INTERFACE ITcoCustomizedDialogFormat

METHOD WithCaption : ITcoCustomizedDialogAnswer
VAR_INPUT
	inCaption : STRING(255);
END_VAR
END_METHOD

METHOD WithImage : ITcoCustomizedDialogAnswer
VAR_INPUT
	inSource : STRING(255);
	inHeight:REAL;
	inWidth:REAL;
END_VAR
END_METHOD

METHOD WithOption1 : ITcoCustomizedDialogAnswer
VAR_INPUT
	inContent:STRING;
END_VAR
END_METHOD

METHOD WithOption2 : ITcoCustomizedDialogAnswer
VAR_INPUT
	inContent:STRING;
END_VAR
END_METHOD

METHOD WithOption3 : ITcoCustomizedDialogAnswer
VAR_INPUT
	inContent:STRING;
END_VAR
END_METHOD

METHOD WithOption4 : ITcoCustomizedDialogAnswer
VAR_INPUT
	inContent:STRING;
END_VAR
END_METHOD

METHOD WithText : ITcoCustomizedDialogAnswer
VAR_INPUT
	inText : STRING(500);
END_VAR
END_METHOD

METHOD WithType : ITcoCustomizedDialogAnswer
VAR_INPUT
	inDialogType : eDialogType;
END_VAR
END_METHOD

END_INTERFACE

(* stored: Version 1.1.0.1
   Itf ITcoCustomizedDialogFormat: Id {1f0fd0b8-9642-0c00-1b66-e7529f799857}
   Folder Format: Id {bd9e39c4-31f1-0f38-04ea-a904b8b6fb6e}
   Method WithCaption: Id {d8b002f1-f8bf-07d7-3800-213a17a3522d}
   Method WithImage: Id {aebba379-3941-0673-304f-e4ee1486f299}
   Method WithOption1: Id {d112fe13-132c-049a-204f-54cbc6221094}
   Method WithOption2: Id {9c314ee7-7606-043b-1b6a-0d81488dc995}
   Method WithOption3: Id {d43c27d8-d80f-074f-2960-0daa9f8a3818}
   Method WithOption4: Id {107a5d45-002e-0221-1076-a8d140d4e744}
   Method WithText: Id {dde53eba-581f-0056-2fc6-776a303264d5}
   Method WithType: Id {876b74e4-01b4-0e68-0e7f-d6f250a2c95d} *)
